// Mitsubishi GX Works2 project: 20141110画像   PLC: FX1N/FX1NC

PROGRAM MAIN
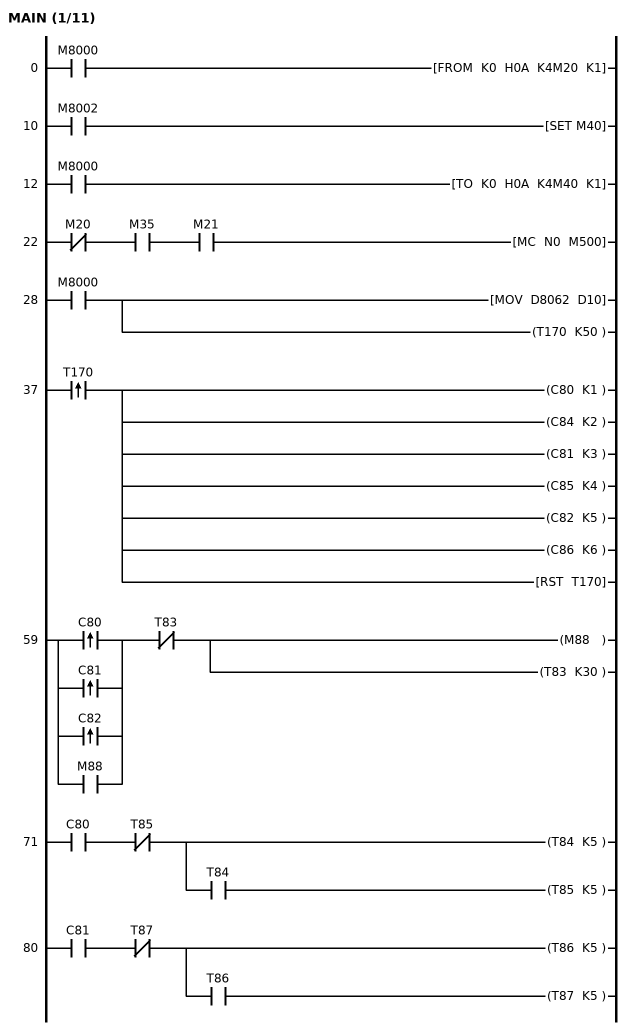
0     LD      M8000
      FROM    K0 H0A K4M20 K1
10    LD      M8002
      SET     M40
12    LD      M8000
      TO      K0 H0A K4M40 K1
22    LDI     M20
      AND     M35
      AND     M21
      MC      N0 M500
28    LD      M8000
      MOV     D8062 D10
      OUT     T170 K50
37    LDP     T170
      OUT     C80 K1
      OUT     C84 K2
      OUT     C81 K3
      OUT     C85 K4
      OUT     C82 K5
      OUT     C86 K6
      RST     T170
59    LDP     C80
      ORP     C81
      ORP     C82
      OR      M88
      ANI     T83
      OUT     M88
      OUT     T83 K30
71    LD      C80
      ANI     T85
      OUT     T84 K5
      AND     T84
      OUT     T85 K5
80    LD      C81
      ANI     T87
      OUT     T86 K5
      AND     T86
      OUT     T87 K5
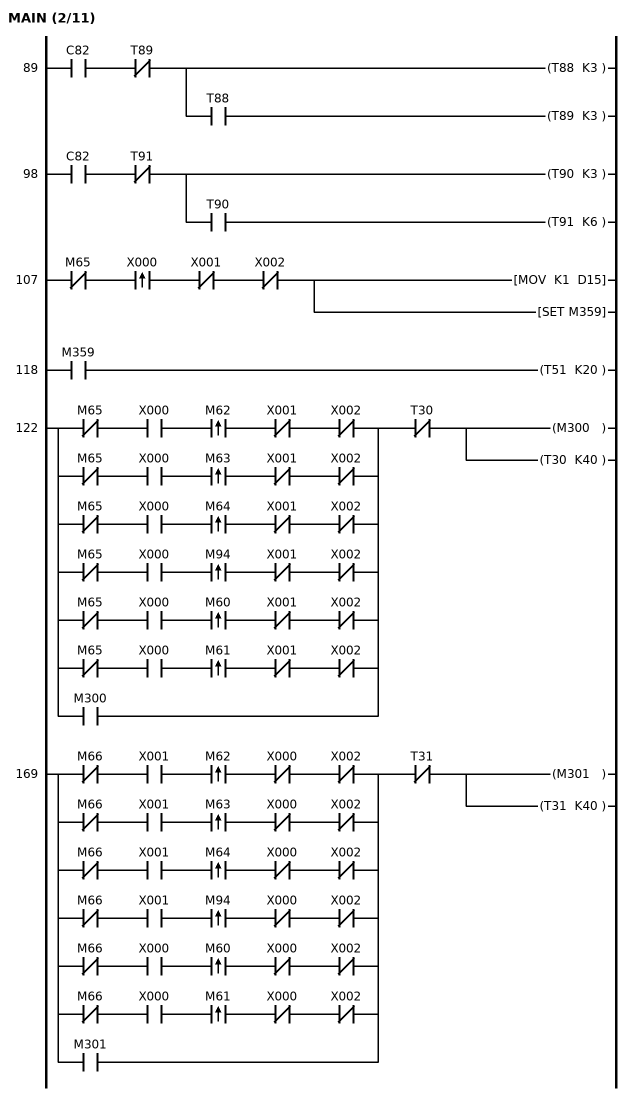
89    LD      C82
      ANI     T89
      OUT     T88 K3
      AND     T88
      OUT     T89 K3
98    LD      C82
      ANI     T91
      OUT     T90 K3
      AND     T90
      OUT     T91 K6
107   LDI     M65
      ANDP    X000
      ANI     X001
      ANI     X002
      MOV     K1 D15
      SET     M359
118   LD      M359
      OUT     T51 K20
122   LDI     M65
      AND     X000
      ANDP    M62
      ANI     X001
      ANI     X002
      LDI     M65
      AND     X000
      ANDP    M63
      ANI     X001
      ANI     X002
      ORB
      LDI     M65
      AND     X000
      ANDP    M64
      ANI     X001
      ANI     X002
      ORB
      LDI     M65
      AND     X000
      ANDP    M94
      ANI     X001
      ANI     X002
      ORB
      LDI     M65
      AND     X000
      ANDP    M60
      ANI     X001
      ANI     X002
      ORB
      LDI     M65
      AND     X000
      ANDP    M61
      ANI     X001
      ANI     X002
      ORB
      OR      M300
      ANI     T30
      OUT     M300
      OUT     T30 K40
169   LDI     M66
      AND     X001
      ANDP    M62
      ANI     X000
      ANI     X002
      LDI     M66
      AND     X001
      ANDP    M63
      ANI     X000
      ANI     X002
      ORB
      LDI     M66
      AND     X001
      ANDP    M64
      ANI     X000
      ANI     X002
      ORB
      LDI     M66
      AND     X001
      ANDP    M94
      ANI     X000
      ANI     X002
      ORB
      LDI     M66
      AND     X000
      ANDP    M60
      ANI     X000
      ANI     X002
      ORB
      LDI     M66
      AND     X000
      ANDP    M61
      ANI     X000
      ANI     X002
      ORB
      OR      M301
      ANI     T31
      OUT     M301
      OUT     T31 K40
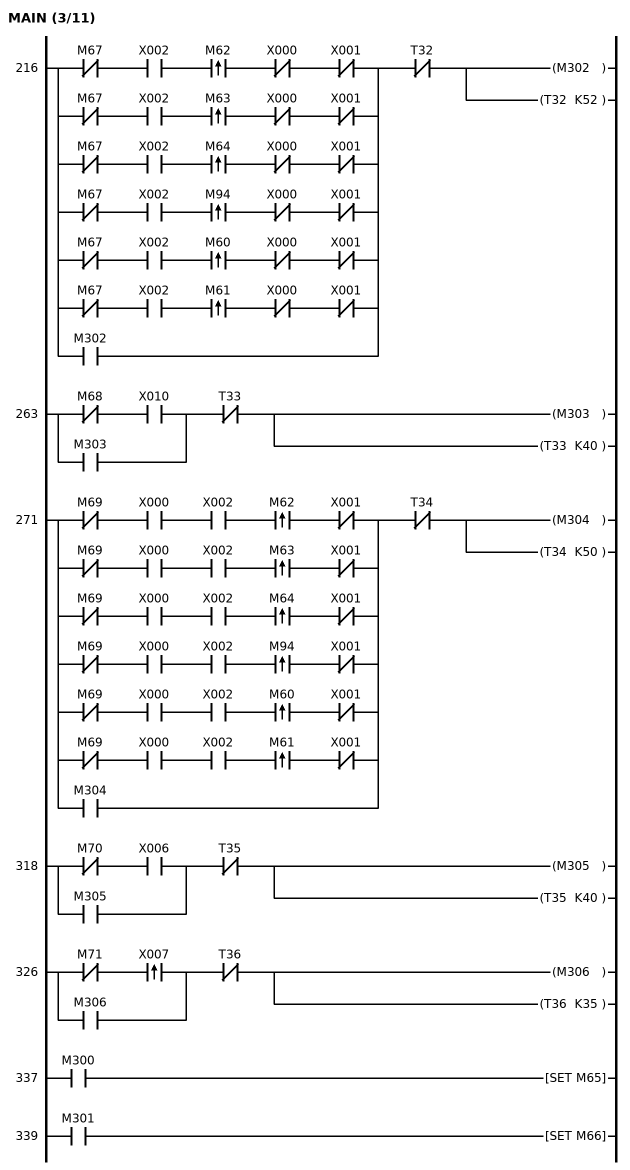
216   LDI     M67
      AND     X002
      ANDP    M62
      ANI     X000
      ANI     X001
      LDI     M67
      AND     X002
      ANDP    M63
      ANI     X000
      ANI     X001
      ORB
      LDI     M67
      AND     X002
      ANDP    M64
      ANI     X000
      ANI     X001
      ORB
      LDI     M67
      AND     X002
      ANDP    M94
      ANI     X000
      ANI     X001
      ORB
      LDI     M67
      AND     X002
      ANDP    M60
      ANI     X000
      ANI     X001
      ORB
      LDI     M67
      AND     X002
      ANDP    M61
      ANI     X000
      ANI     X001
      ORB
      OR      M302
      ANI     T32
      OUT     M302
      OUT     T32 K52
263   LDI     M68
      AND     X010
      OR      M303
      ANI     T33
      OUT     M303
      OUT     T33 K40
271   LDI     M69
      AND     X000
      AND     X002
      ANDP    M62
      ANI     X001
      LDI     M69
      AND     X000
      AND     X002
      ANDP    M63
      ANI     X001
      ORB
      LDI     M69
      AND     X000
      AND     X002
      ANDP    M64
      ANI     X001
      ORB
      LDI     M69
      AND     X000
      AND     X002
      ANDP    M94
      ANI     X001
      ORB
      LDI     M69
      AND     X000
      AND     X002
      ANDP    M60
      ANI     X001
      ORB
      LDI     M69
      AND     X000
      AND     X002
      ANDP    M61
      ANI     X001
      ORB
      OR      M304
      ANI     T34
      OUT     M304
      OUT     T34 K50
318   LDI     M70
      AND     X006
      OR      M305
      ANI     T35
      OUT     M305
      OUT     T35 K40
326   LDI     M71
      ANDP    X007
      OR      M306
      ANI     T36
      OUT     M306
      OUT     T36 K35
337   LD      M300
      SET     M65
339   LD      M301
      SET     M66
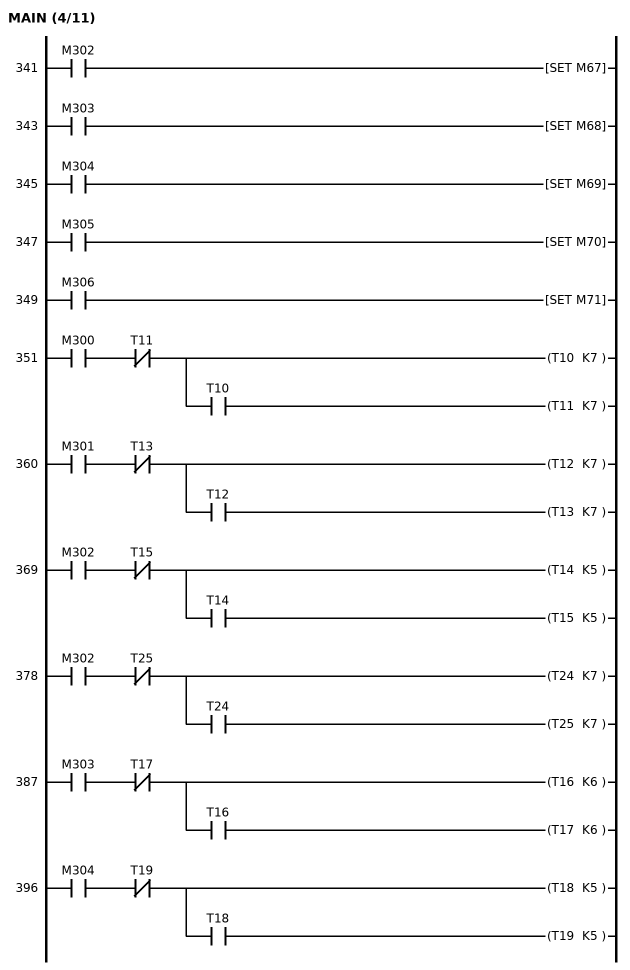
341   LD      M302
      SET     M67
343   LD      M303
      SET     M68
345   LD      M304
      SET     M69
347   LD      M305
      SET     M70
349   LD      M306
      SET     M71
351   LD      M300
      ANI     T11
      OUT     T10 K7
      AND     T10
      OUT     T11 K7
360   LD      M301
      ANI     T13
      OUT     T12 K7
      AND     T12
      OUT     T13 K7
369   LD      M302
      ANI     T15
      OUT     T14 K5
      AND     T14
      OUT     T15 K5
378   LD      M302
      ANI     T25
      OUT     T24 K7
      AND     T24
      OUT     T25 K7
387   LD      M303
      ANI     T17
      OUT     T16 K6
      AND     T16
      OUT     T17 K6
396   LD      M304
      ANI     T19
      OUT     T18 K5
      AND     T18
      OUT     T19 K5
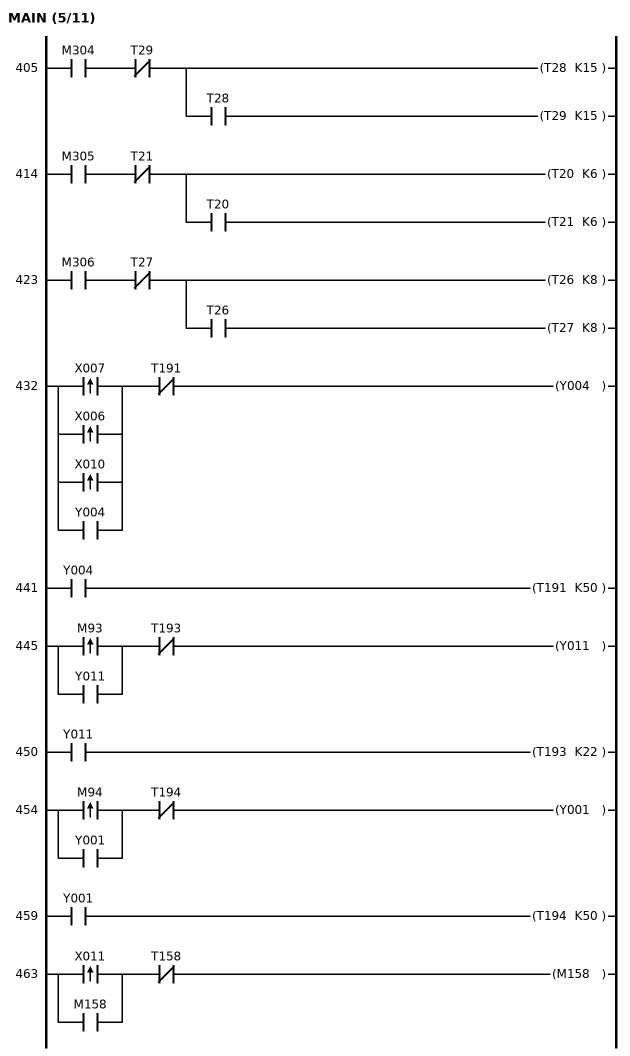
405   LD      M304
      ANI     T29
      OUT     T28 K15
      AND     T28
      OUT     T29 K15
414   LD      M305
      ANI     T21
      OUT     T20 K6
      AND     T20
      OUT     T21 K6
423   LD      M306
      ANI     T27
      OUT     T26 K8
      AND     T26
      OUT     T27 K8
432   LDP     X007
      ORP     X006
      ORP     X010
      OR      Y004
      ANI     T191
      OUT     Y004
441   LD      Y004
      OUT     T191 K50
445   LDP     M93
      OR      Y011
      ANI     T193
      OUT     Y011
450   LD      Y011
      OUT     T193 K22
454   LDP     M94
      OR      Y001
      ANI     T194
      OUT     Y001
459   LD      Y001
      OUT     T194 K50
463   LDP     X011
      OR      M158
      ANI     T158
      OUT     M158
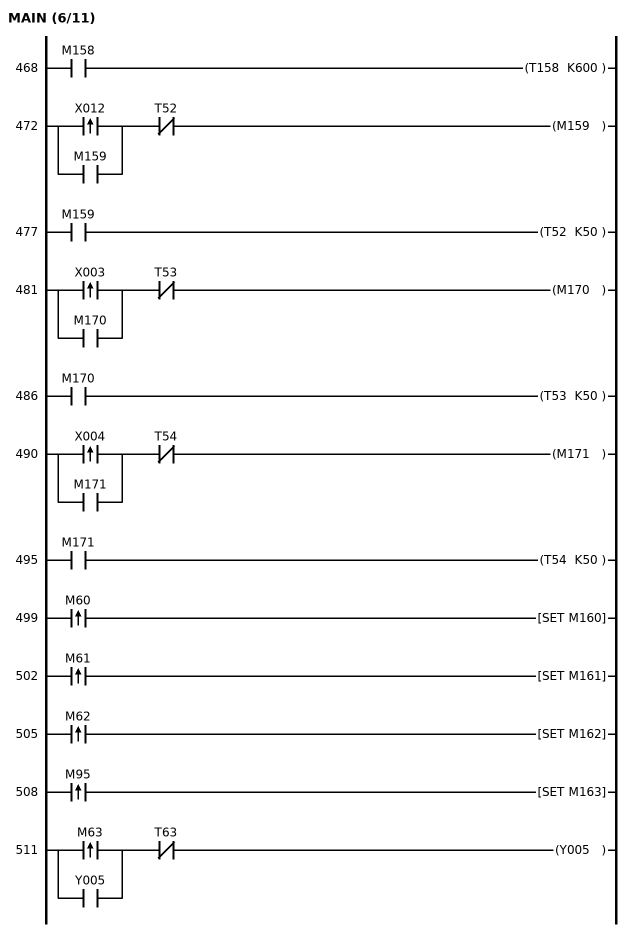
468   LD      M158
      OUT     T158 K600
472   LDP     X012
      OR      M159
      ANI     T52
      OUT     M159
477   LD      M159
      OUT     T52 K50
481   LDP     X003
      OR      M170
      ANI     T53
      OUT     M170
486   LD      M170
      OUT     T53 K50
490   LDP     X004
      OR      M171
      ANI     T54
      OUT     M171
495   LD      M171
      OUT     T54 K50
499   LDP     M60
      SET     M160
502   LDP     M61
      SET     M161
505   LDP     M62
      SET     M162
508   LDP     M95
      SET     M163
511   LDP     M63
      OR      Y005
      ANI     T63
      OUT     Y005
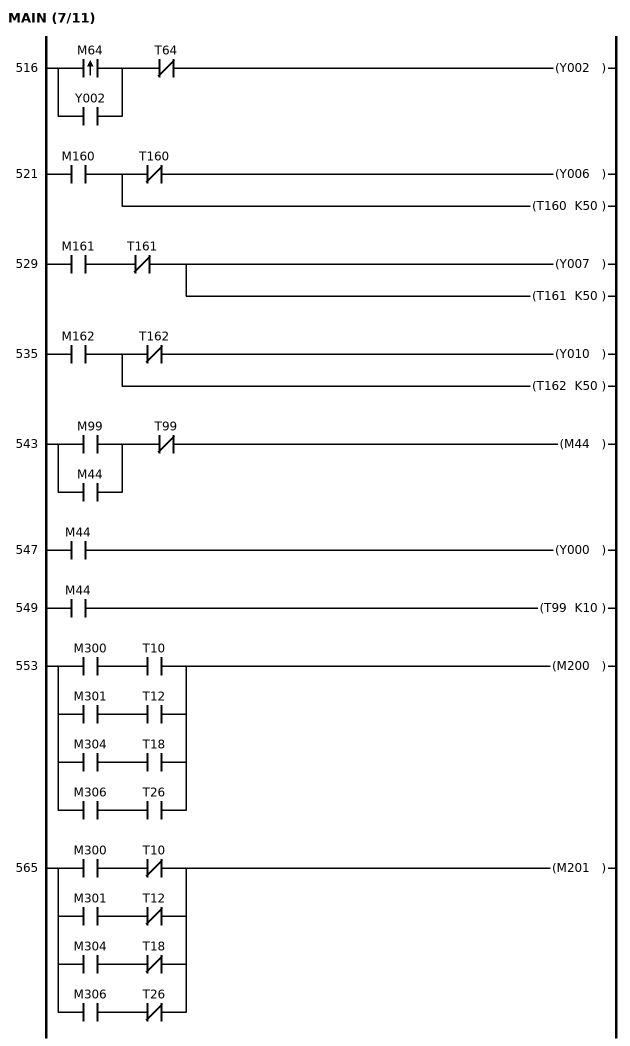
516   LDP     M64
      OR      Y002
      ANI     T64
      OUT     Y002
521   LD      M160
      MPS
      ANI     T160
      OUT     Y006
      MPP
      OUT     T160 K50
529   LD      M161
      ANI     T161
      OUT     Y007
      OUT     T161 K50
535   LD      M162
      MPS
      ANI     T162
      OUT     Y010
      MPP
      OUT     T162 K50
543   LD      M99
      OR      M44
      ANI     T99
      OUT     M44
547   LD      M44
      OUT     Y000
549   LD      M44
      OUT     T99 K10
553   LD      M300
      AND     T10
      LD      M301
      AND     T12
      ORB
      LD      M304
      AND     T18
      ORB
      LD      M306
      AND     T26
      ORB
      OUT     M200
565   LD      M300
      ANI     T10
      LD      M301
      ANI     T12
      ORB
      LD      M304
      ANI     T18
      ORB
      LD      M306
      ANI     T26
      ORB
      OUT     M201
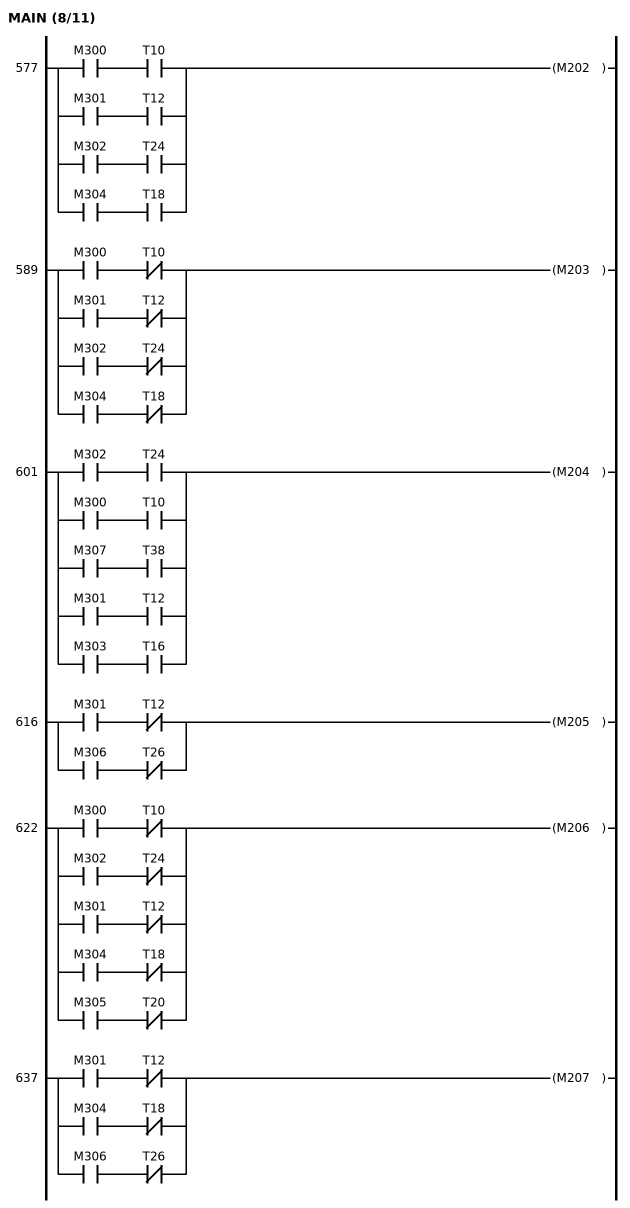
577   LD      M300
      AND     T10
      LD      M301
      AND     T12
      ORB
      LD      M302
      AND     T24
      ORB
      LD      M304
      AND     T18
      ORB
      OUT     M202
589   LD      M300
      ANI     T10
      LD      M301
      ANI     T12
      ORB
      LD      M302
      ANI     T24
      ORB
      LD      M304
      ANI     T18
      ORB
      OUT     M203
601   LD      M302
      AND     T24
      LD      M300
      AND     T10
      ORB
      LD      M307
      AND     T38
      ORB
      LD      M301
      AND     T12
      ORB
      LD      M303
      AND     T16
      ORB
      OUT     M204
616   LD      M301
      ANI     T12
      LD      M306
      ANI     T26
      ORB
      OUT     M205
622   LD      M300
      ANI     T10
      LD      M302
      ANI     T24
      ORB
      LD      M301
      ANI     T12
      ORB
      LD      M304
      ANI     T18
      ORB
      LD      M305
      ANI     T20
      ORB
      OUT     M206
637   LD      M301
      ANI     T12
      LD      M304
      ANI     T18
      ORB
      LD      M306
      ANI     T26
      ORB
      OUT     M207
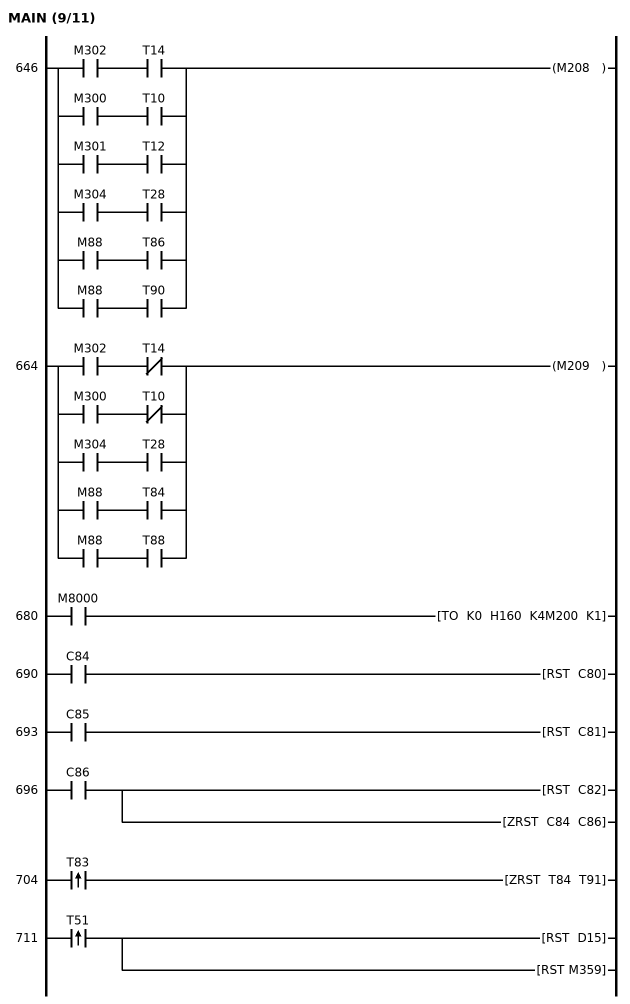
646   LD      M302
      AND     T14
      LD      M300
      AND     T10
      ORB
      LD      M301
      AND     T12
      ORB
      LD      M304
      AND     T28
      ORB
      LD      M88
      AND     T86
      ORB
      LD      M88
      AND     T90
      ORB
      OUT     M208
664   LD      M302
      ANI     T14
      LD      M300
      ANI     T10
      ORB
      LD      M304
      AND     T28
      ORB
      LD      M88
      AND     T84
      ORB
      LD      M88
      AND     T88
      ORB
      OUT     M209
680   LD      M8000
      TO      K0 H160 K4M200 K1
690   LD      C84
      RST     C80
693   LD      C85
      RST     C81
696   LD      C86
      RST     C82
      ZRST    C84 C86
704   LDP     T83
      ZRST    T84 T91
711   LDP     T51
      RST     D15
      RST     M359
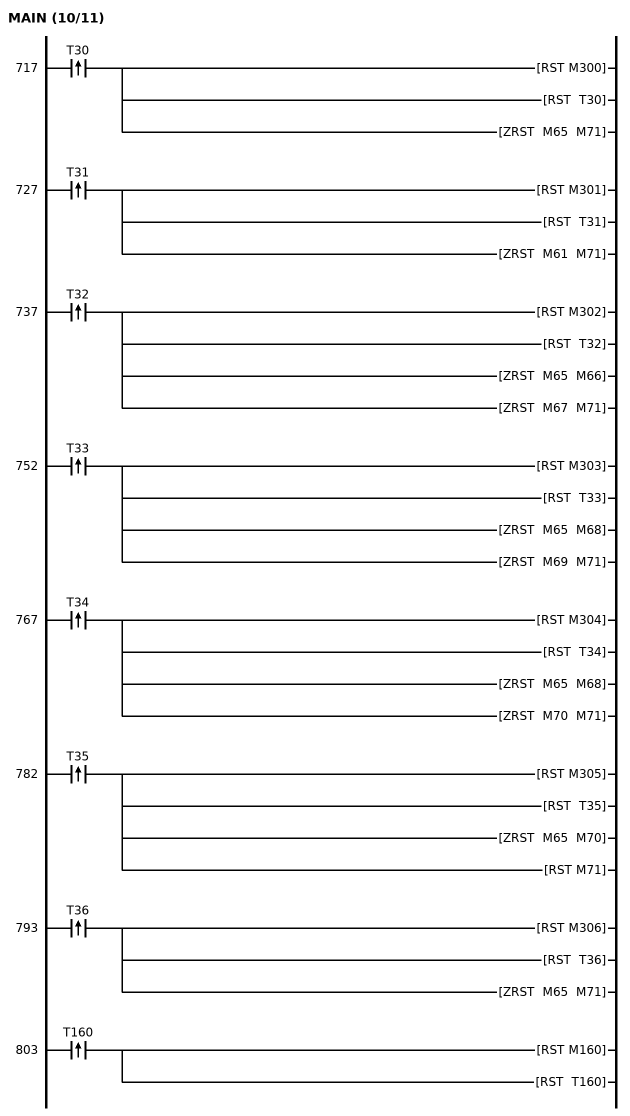
717   LDP     T30
      RST     M300
      RST     T30
      ZRST    M65 M71
727   LDP     T31
      RST     M301
      RST     T31
      ZRST    M61 M71
737   LDP     T32
      RST     M302
      RST     T32
      ZRST    M65 M66
      ZRST    M67 M71
752   LDP     T33
      RST     M303
      RST     T33
      ZRST    M65 M68
      ZRST    M69 M71
767   LDP     T34
      RST     M304
      RST     T34
      ZRST    M65 M68
      ZRST    M70 M71
782   LDP     T35
      RST     M305
      RST     T35
      ZRST    M65 M70
      RST     M71
793   LDP     T36
      RST     M306
      RST     T36
      ZRST    M65 M71
803   LDP     T160
      RST     M160
      RST     T160
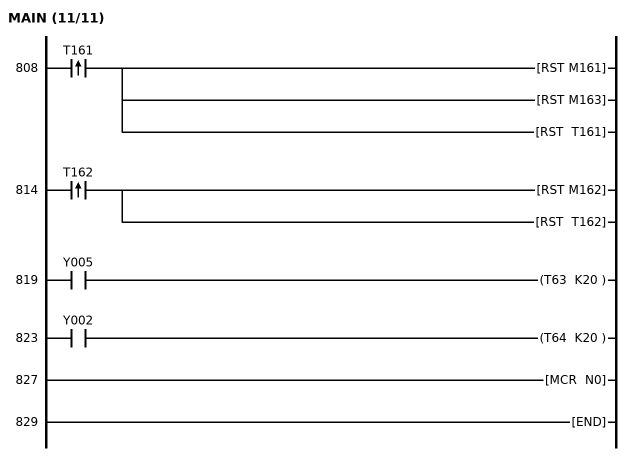
808   LDP     T161
      RST     M161
      RST     M163
      RST     T161
814   LDP     T162
      RST     M162
      RST     T162
819   LD      Y005
      OUT     T63 K20
823   LD      Y002
      OUT     T64 K20
827   MCR     N0
829   END
END_PROGRAM
